// TIA Portal V19 export
DATA_BLOCK "PG_Devices"   // DB28
{ S7_Optimized_Access := 'TRUE' }
// stored: AutoNumber false, MemoryReserve 0
   VAR RETAIN
      V0552 : "IO Burkett Type 8691 r3";
      V0934 : "IO Burkett Type 8691 r3";
      V0935 : "IO Burkett Type 8691 r3";
      DI_100_005_X06_X1_3p4 : Bool;   // PN_100, Node 5, Port 6 X1.3 pin4 - GS09.40
      DI_100_005_X06_X1_3p2 : Bool;   // PN_100, Node 5, Port 6 X1.3 pin2 - GS09.41
      V0940 : "TetraPakV50_IO";
      V0941 : "TetraPakV50_IO";
      V0942 : "TetraPakV50_IO";
      V0943 : "TetraPakV50_IO";
      V0944 : "TetraPakV50_IO";
      TTX0940 : "IFM_TA1612_IO";
      TTX0941 : "IFM_TA1612_IO";
      TTX0942 : "IFM_TA1612_IO";
      PTX0940 : "IFM_PI1714_IO";
      PTX0941 : "IFM_PI1714_IO";
      CTX0931 : "IFM_LDL_IO";
      V0945_SV1 : Bool;
      V0945_SV2 : Bool;
      V0945_Open : Bool;
      V0945_Closed : Bool;
      M0940_Iso : Bool;
      M0941_Iso : Bool;
      V0945_pa_auto_req : Bool;   // Pressure Assist - SV2 request
      V1021 : "TetraPakV70_IO";
      V1023 : "TetraPakV50_IO";
      V1024 : "IO Burkett Type 8691 r3";
      V1025 : "TetraPakV50_IO";
      V1027 : "TetraPakV50_IO";
      V1083 : "TetraPakV50_IO";
      TTX1040 : "IFM_TA1612_IO";
      TTX1041 : "IFM_TA1612_IO";
      DI_100_012_X1_1p4 : Bool;   // PN 100, Node 12, X1.1p4 - EmptyLine Pushbutton
      DO_100_012_X1_2p4 : Bool;   // PN 100, Node 12, X1.2p4 - EOL in use Beacon
      DI_100_010_X01_4 : Bool;   // PN 100, Node 10, X01.4 - M09.40 MPCB Tripped
      DI_100_010_X02_4 : Bool;   // PN 100, Node 10, X02.4 - M09.41 Run
      DI_100_010_X03_4 : Bool;   // PN 100, Node 10, X03.4 - M09.41 MPCB Tripped
      DO_100_010_X04_4 : Bool;   // PN 100, Node 10, X04.4 - M09.41 Req
      DO_100_012_X1_0p4 : Bool;   // PN 100, Node 12, X1.0p4 - Polygon F2 Product at Filler
      FT0940 : "EH_ProMag300_PD_UDT";
      LS1074 : "IFM LMT100_IO";
      TTX0940_Params : "IF_TA1612_TTxNest";   // Acyclic parameter read/write
      TTX0941_Params : "IF_TA1612_TTxNest";   // Acyclic parameter read/write
      TTX0942_Params : "IF_TA1612_TTxNest";   // Acyclic parameter read/write
      TTX1040_Params : "IF_TA1612_TTxNest";   // Acyclic parameter read/write
      TTX1041_Params : "IF_TA1612_TTxNest";   // Acyclic parameter read/write
      V0552_Params : "BurkettType8691_UDTNest";
      V0934_Params : "BurkettType8691_UDTNest";
      V0935_Params : "BurkettType8691_UDTNest";
      V0940_Params : "TetraPakV50_9_UDTNest";
      V0941_Params : "TetraPakV50_9_UDTNest";
      V0942_Params : "TetraPakV50_9_UDTNest";
      V0943_Params : "TetraPakV50_9_UDTNest";
      V0944_Params : "TetraPakV50_9_UDTNest";
      V1021_Params : "TetraPakV70_10_UDTNest";
      V1023_Params : "TetraPakV50_9_UDTNest";
      V1024_Params : "BurkettType8691_UDTNest";
      V1025_Params : "TetraPakV50_9_UDTNest";
      V1027_Params : "TetraPakV50_9_UDTNest";
      V1083_Params : "TetraPakV50_9_UDTNest";
      DI_100_012_X1_1p2 : Bool;   // PN_100, Node 12, X1.1p2 - PG_EOL_CS
      CTX2274 : "IFM_LDL_IO";
      V0936 : "TetraPakV50_IO";
      V0936_Params : "TetraPakV50_9_UDTNest";
      PTX0945 : "IFM_PN3594_IO";
   END_VAR
BEGIN
   V0552.OUT.ValvePosition := 0.0;
   V0934.OUT.ValvePosition := 0.0;
   V0935.OUT.ValvePosition := 0.0;
   V0940.OUT.ValvePosition := 0.0;
   V0941.OUT.ValvePosition := 0.0;
   V0942.OUT.ValvePosition := 0.0;
   V0943.OUT.ValvePosition := 0.0;
   V0944.OUT.ValvePosition := 0.0;
   TTX0940.Addr := 426;
   TTX0940.Value := 0.0;
   TTX0941.Value := 0.0;
   TTX0942.Value := 0.0;
   PTX0940.Value_p := 0.0;
   PTX0940.Value_t := 0.0;
   PTX0941.Value_p := 0.0;
   PTX0941.Value_t := 0.0;
   CTX0931.Value_c := 0.0;
   CTX0931.Value_t := 0.0;
   V1021.OUT.ValvePosition := 0.0;
   V1023.OUT.ValvePosition := 0.0;
   V1024.OUT.ValvePosition := 0.0;
   V1025.OUT.ValvePosition := 0.0;
   V1027.OUT.ValvePosition := 0.0;
   V1083.OUT.ValvePosition := 0.0;
   TTX1040.Value := 0.0;
   TTX1041.Value := 0.0;
   FT0940.Volume_Flow := 0.0;
   FT0940.Totaliser_Value := 0.0;
   TTX0940_Params.OP.I_DataStorage := TRUE;
   TTX0940_Params.OP.I_BlockParam := TRUE;
   TTX0941_Params.OP.I_DataStorage := TRUE;
   TTX0941_Params.OP.I_BlockParam := TRUE;
   TTX0942_Params.OP.I_DataStorage := TRUE;
   TTX0942_Params.OP.I_BlockParam := TRUE;
   TTX1040_Params.OP.I_DataStorage := TRUE;
   TTX1040_Params.OP.I_BlockParam := TRUE;
   TTX1041_Params.OP.I_DataStorage := TRUE;
   TTX1041_Params.OP.I_BlockParam := TRUE;
   V0552_Params."IF".StandardStructure.DeviceParameters.Parameter_05.Value.ProgressTotaliser := 0.0;
   V0552_Params."IF".StandardStructure.DeviceParameters.Parameter_06.Value.IntervalTotaliser := 0.0;
   V0552_Params."IF".StandardStructure.DeviceParameters.Parameter_07.Value.ValueTotaliser := 0.0;
   V0552_Params."IF".StandardStructure.DeviceParameters.Parameter_08.Value.EnableTotaliser := B#16#0;
   V0552_Params."IF".StandardStructure.DeviceParameters.Parameter_10.Value.ProgressTotaliser := 0.0;
   V0552_Params."IF".StandardStructure.DeviceParameters.Parameter_14.Value.ProgressTotaliser := 0.0;
   V0934_Params."IF".StandardStructure.DeviceParameters.Parameter_05.Value.ProgressTotaliser := 0.0;
   V0934_Params."IF".StandardStructure.DeviceParameters.Parameter_06.Value.IntervalTotaliser := 0.0;
   V0934_Params."IF".StandardStructure.DeviceParameters.Parameter_07.Value.ValueTotaliser := 0.0;
   V0934_Params."IF".StandardStructure.DeviceParameters.Parameter_10.Value.ProgressTotaliser := 0.0;
   V0934_Params."IF".StandardStructure.DeviceParameters.Parameter_14.Value.ProgressTotaliser := 0.0;
   V0935_Params."IF".StandardStructure.DeviceParameters.Parameter_05.Value.ProgressTotaliser := 0.0;
   V0935_Params."IF".StandardStructure.DeviceParameters.Parameter_06.Value.IntervalTotaliser := 0.0;
   V0935_Params."IF".StandardStructure.DeviceParameters.Parameter_07.Value.ValueTotaliser := 0.0;
   V0935_Params."IF".StandardStructure.DeviceParameters.Parameter_10.Value.ProgressTotaliser := 0.0;
   V0935_Params."IF".StandardStructure.DeviceParameters.Parameter_14.Value.ProgressTotaliser := 0.0;
   V0940_Params.OP.I_DataStorage := TRUE;
   V0940_Params.OP.I_BlockParam := TRUE;
   V0940_Params."IF".StandardStructure.DeviceIndentification.V_FirmwareRevision.Length := 5;
   V0941_Params.OP.I_DataStorage := TRUE;
   V0941_Params.OP.I_BlockParam := TRUE;
   V0942_Params.OP.I_DataStorage := TRUE;
   V0942_Params.OP.I_BlockParam := TRUE;
   V0943_Params.OP.I_DataStorage := TRUE;
   V0943_Params.OP.I_BlockParam := TRUE;
   V0944_Params.OP.I_DataStorage := TRUE;
   V0944_Params.OP.I_BlockParam := TRUE;
   V1021_Params.OP.I_DataStorage := TRUE;
   V1021_Params.OP.I_BlockParam := TRUE;
   V1023_Params.OP.I_DataStorage := TRUE;
   V1023_Params.OP.I_BlockParam := TRUE;
   V1023_Params."IF".StandardStructure.Commando.Commando_04.IOLStat := DWORD#16#0000_1023;
   V1024_Params."IF".StandardStructure.DeviceParameters.Parameter_05.Value.ProgressTotaliser := 0.0;
   V1024_Params."IF".StandardStructure.DeviceParameters.Parameter_06.Value.IntervalTotaliser := 0.0;
   V1024_Params."IF".StandardStructure.DeviceParameters.Parameter_07.Value.ValueTotaliser := 0.0;
   V1024_Params."IF".StandardStructure.DeviceParameters.Parameter_10.Value.ProgressTotaliser := 0.0;
   V1024_Params."IF".StandardStructure.DeviceParameters.Parameter_14.Value.ProgressTotaliser := 0.0;
   V1025_Params.OP.I_DataStorage := TRUE;
   V1025_Params.OP.I_BlockParam := TRUE;
   V1025_Params."IF".StandardStructure.Commando.Commando_04.IOLStat := DWORD#16#0001_0237;
   V1027_Params.OP.I_DataStorage := TRUE;
   V1027_Params.OP.I_BlockParam := TRUE;
   V1027_Params."IF".StandardStructure.Commando.Commando_04.IOLStat := DWORD#16#0001_0283;
   V1083_Params.OP.I_DataStorage := TRUE;
   V1083_Params.OP.I_BlockParam := TRUE;
   V1083_Params."IF".StandardStructure.Commando.Commando_04.IOLStat := DWORD#16#0000_1023;
   CTX2274.Value_c := 0.0;
   CTX2274.Value_t := 0.0;
   V0936.OUT.ValvePosition := 0.0;
   PTX0945.Value := 0.0;
END_DATA_BLOCK
